# EPICS substitutions: iocBoot/iocAMControls/amControls.substitutions
file "$(TOP)/db/amControls.template"
{
pattern
{  P,        R,      CAMERA_PREFIX,   EXAMPLE_PV_NAME}
{32id:, AMControls:,    2bmbSP2:      32id:m1}
}
